{attribute 'qualified_only'}
{attribute 'strict'}
TYPE E_InfluxReaderState :
(
	Idle := 0,
	Connecting,
	Query,
	ConvertingNumbers, 
	Disconnecting
) DINT;
END_TYPE

(* stored: Version 1.1.0.1, ProductVersion 3.1.4022.11
   DUT E_InfluxReaderState: Id {89da615a-9188-4bf9-955a-d9dfdadeed33} *)
